    ! Character: ^
    PROC char_caret(\num nScaleParam)
        VAR robtarget pTarget;
        VAR num nScale:=1;
        pTarget:=refTarget;
        IF Present(nScaleParam) THEN
            nScale:=nScaleParam;
        ENDIF
        pTarget.trans:=[8*nScale,34.0*nScale,0];
        MoveL pTarget,vSpeed,fine,tTool\WObj:=wWobj;
        Set do_pen;
        pTarget.trans:=[0*nScale,20.0*nScale,0];
        MoveL pTarget,vSpeed,fine,tTool\WObj:=wWobj;
        Reset do_pen;
        MoveL RelTool(pTarget,0,0,-2),vSpeed,z0,tTool\WObj:=wWobj;
        pTarget.trans:=[8*nScale,34.0*nScale,0];
        MoveL pTarget,vSpeed,fine,tTool\WObj:=wWobj;
        Set do_pen;
        pTarget.trans:=[16*nScale,20.0*nScale,0];
        MoveL pTarget,vSpeed,fine,tTool\WObj:=wWobj;
        Reset do_pen;
        MoveL RelTool(pTarget,0,0,-2),vSpeed,z0,tTool\WObj:=wWobj;
        wWobj.oframe.trans.x:=wWobj.oframe.trans.x+16*nScale;
    ENDPROC

    ! Character: &
    PROC char_ampersand(\num nScaleParam)
        VAR robtarget pTarget;
        VAR num nScale:=1;
        pTarget:=refTarget;
        IF Present(nScaleParam) THEN
            nScale:=nScaleParam;
        ENDIF
        pTarget.trans:=[23*nScale,23.0*nScale,0];
        MoveL pTarget,vSpeed,fine,tTool\WObj:=wWobj;
        Set do_pen;
        pTarget.trans:=[23*nScale,24.0*nScale,0];
        MoveL pTarget,vSpeed,z0,tTool\WObj:=wWobj;
        pTarget.trans:=[22*nScale,25.0*nScale,0];
        MoveL pTarget,vSpeed,z0,tTool\WObj:=wWobj;
        pTarget.trans:=[21*nScale,25.0*nScale,0];
        MoveL pTarget,vSpeed,z0,tTool\WObj:=wWobj;
        pTarget.trans:=[20*nScale,24.0*nScale,0];
        MoveL pTarget,vSpeed,z0,tTool\WObj:=wWobj;
        pTarget.trans:=[19*nScale,22.0*nScale,0];
        MoveL pTarget,vSpeed,z0,tTool\WObj:=wWobj;
        pTarget.trans:=[17*nScale,17.0*nScale,0];
        MoveL pTarget,vSpeed,z0,tTool\WObj:=wWobj;
        pTarget.trans:=[15*nScale,14.0*nScale,0];
        MoveL pTarget,vSpeed,z0,tTool\WObj:=wWobj;
        pTarget.trans:=[13*nScale,12.0*nScale,0];
        MoveL pTarget,vSpeed,z0,tTool\WObj:=wWobj;
        pTarget.trans:=[11*nScale,11.0*nScale,0];
        MoveL pTarget,vSpeed,z0,tTool\WObj:=wWobj;
        pTarget.trans:=[7*nScale,11.0*nScale,0];
        MoveL pTarget,vSpeed,z0,tTool\WObj:=wWobj;
        pTarget.trans:=[5*nScale,12.0*nScale,0];
        MoveL pTarget,vSpeed,z0,tTool\WObj:=wWobj;
        pTarget.trans:=[4*nScale,13.0*nScale,0];
        MoveL pTarget,vSpeed,z0,tTool\WObj:=wWobj;
        pTarget.trans:=[3*nScale,15.0*nScale,0];
        MoveL pTarget,vSpeed,z0,tTool\WObj:=wWobj;
        pTarget.trans:=[3*nScale,17.0*nScale,0];
        MoveL pTarget,vSpeed,z0,tTool\WObj:=wWobj;
        pTarget.trans:=[4*nScale,19.0*nScale,0];
        MoveL pTarget,vSpeed,z0,tTool\WObj:=wWobj;
        pTarget.trans:=[5*nScale,20.0*nScale,0];
        MoveL pTarget,vSpeed,z0,tTool\WObj:=wWobj;
        pTarget.trans:=[12*nScale,24.0*nScale,0];
        MoveL pTarget,vSpeed,z0,tTool\WObj:=wWobj;
        pTarget.trans:=[13*nScale,25.0*nScale,0];
        MoveL pTarget,vSpeed,z0,tTool\WObj:=wWobj;
        pTarget.trans:=[14*nScale,27.0*nScale,0];
        MoveL pTarget,vSpeed,z0,tTool\WObj:=wWobj;
        pTarget.trans:=[14*nScale,29.0*nScale,0];
        MoveL pTarget,vSpeed,z0,tTool\WObj:=wWobj;
        pTarget.trans:=[13*nScale,31.0*nScale,0];
        MoveL pTarget,vSpeed,z0,tTool\WObj:=wWobj;
        pTarget.trans:=[11*nScale,32.0*nScale,0];
        MoveL pTarget,vSpeed,z0,tTool\WObj:=wWobj;
        pTarget.trans:=[9*nScale,31.0*nScale,0];
        MoveL pTarget,vSpeed,z0,tTool\WObj:=wWobj;
        pTarget.trans:=[8*nScale,29.0*nScale,0];
        MoveL pTarget,vSpeed,z0,tTool\WObj:=wWobj;
        pTarget.trans:=[8*nScale,27.0*nScale,0];
        MoveL pTarget,vSpeed,z0,tTool\WObj:=wWobj;
        pTarget.trans:=[9*nScale,24.0*nScale,0];
        MoveL pTarget,vSpeed,z0,tTool\WObj:=wWobj;
        pTarget.trans:=[11*nScale,21.0*nScale,0];
        MoveL pTarget,vSpeed,z0,tTool\WObj:=wWobj;
        pTarget.trans:=[16*nScale,14.0*nScale,0];
        MoveL pTarget,vSpeed,z0,tTool\WObj:=wWobj;
        pTarget.trans:=[18*nScale,12.0*nScale,0];
        MoveL pTarget,vSpeed,z0,tTool\WObj:=wWobj;
        pTarget.trans:=[20*nScale,11.0*nScale,0];
        MoveL pTarget,vSpeed,z0,tTool\WObj:=wWobj;
        pTarget.trans:=[22*nScale,11.0*nScale,0];
        MoveL pTarget,vSpeed,z0,tTool\WObj:=wWobj;
        pTarget.trans:=[23*nScale,12.0*nScale,0];
        MoveL pTarget,vSpeed,z0,tTool\WObj:=wWobj;
        pTarget.trans:=[23*nScale,13.0*nScale,0];
        MoveL pTarget,vSpeed,fine,tTool\WObj:=wWobj;
        Reset do_pen;
        MoveL RelTool(pTarget,0,0,-2),vSpeed,z0,tTool\WObj:=wWobj;
        wWobj.oframe.trans.x:=wWobj.oframe.trans.x+26*nScale;
    ENDPROC

    ! Character: *
    PROC char_asterisk(\num nScaleParam)
        VAR robtarget pTarget;
        VAR num nScale:=1;
        pTarget:=refTarget;
        IF Present(nScaleParam) THEN
            nScale:=nScaleParam;
        ENDIF
        pTarget.trans:=[8*nScale,26.0*nScale,0];
        MoveL pTarget,vSpeed,fine,tTool\WObj:=wWobj;
        Set do_pen;
        pTarget.trans:=[8*nScale,14.0*nScale,0];
        MoveL pTarget,vSpeed,fine,tTool\WObj:=wWobj;
        Reset do_pen;
        MoveL RelTool(pTarget,0,0,-2),vSpeed,z0,tTool\WObj:=wWobj;
        pTarget.trans:=[3*nScale,23.0*nScale,0];
        MoveL pTarget,vSpeed,fine,tTool\WObj:=wWobj;
        Set do_pen;
        pTarget.trans:=[13*nScale,17.0*nScale,0];
        MoveL pTarget,vSpeed,fine,tTool\WObj:=wWobj;
        Reset do_pen;
        MoveL RelTool(pTarget,0,0,-2),vSpeed,z0,tTool\WObj:=wWobj;
        pTarget.trans:=[13*nScale,23.0*nScale,0];
        MoveL pTarget,vSpeed,fine,tTool\WObj:=wWobj;
        Set do_pen;
        pTarget.trans:=[3*nScale,17.0*nScale,0];
        MoveL pTarget,vSpeed,fine,tTool\WObj:=wWobj;
        Reset do_pen;
        MoveL RelTool(pTarget,0,0,-2),vSpeed,z0,tTool\WObj:=wWobj;
        wWobj.oframe.trans.x:=wWobj.oframe.trans.x+16*nScale;
    ENDPROC

    ! Character: (
    PROC char_leftparenthesis(\num nScaleParam)
        VAR robtarget pTarget;
        VAR num nScale:=1;
        pTarget:=refTarget;
        IF Present(nScaleParam) THEN
            nScale:=nScaleParam;
        ENDIF
        pTarget.trans:=[11*nScale,36.0*nScale,0];
        MoveL pTarget,vSpeed,fine,tTool\WObj:=wWobj;
        Set do_pen;
        pTarget.trans:=[9*nScale,34.0*nScale,0];
        MoveL pTarget,vSpeed,z0,tTool\WObj:=wWobj;
        pTarget.trans:=[7*nScale,31.0*nScale,0];
        MoveL pTarget,vSpeed,z0,tTool\WObj:=wWobj;
        pTarget.trans:=[5*nScale,27.0*nScale,0];
        MoveL pTarget,vSpeed,z0,tTool\WObj:=wWobj;
        pTarget.trans:=[4*nScale,22.0*nScale,0];
        MoveL pTarget,vSpeed,z0,tTool\WObj:=wWobj;
        pTarget.trans:=[4*nScale,18.0*nScale,0];
        MoveL pTarget,vSpeed,z0,tTool\WObj:=wWobj;
        pTarget.trans:=[5*nScale,13.0*nScale,0];
        MoveL pTarget,vSpeed,z0,tTool\WObj:=wWobj;
        pTarget.trans:=[7*nScale,9.0*nScale,0];
        MoveL pTarget,vSpeed,z0,tTool\WObj:=wWobj;
        pTarget.trans:=[9*nScale,6.0*nScale,0];
        MoveL pTarget,vSpeed,z0,tTool\WObj:=wWobj;
        pTarget.trans:=[11*nScale,4.0*nScale,0];
        MoveL pTarget,vSpeed,fine,tTool\WObj:=wWobj;
        Reset do_pen;
        MoveL RelTool(pTarget,0,0,-2),vSpeed,z0,tTool\WObj:=wWobj;
        wWobj.oframe.trans.x:=wWobj.oframe.trans.x+14*nScale;
    ENDPROC

    ! Character: )
    PROC char_rightparenthesis(\num nScaleParam)
        VAR robtarget pTarget;
        VAR num nScale:=1;
        pTarget:=refTarget;
        IF Present(nScaleParam) THEN
            nScale:=nScaleParam;
        ENDIF
        pTarget.trans:=[3*nScale,36.0*nScale,0];
        MoveL pTarget,vSpeed,fine,tTool\WObj:=wWobj;
        Set do_pen;
        pTarget.trans:=[5*nScale,34.0*nScale,0];
        MoveL pTarget,vSpeed,z0,tTool\WObj:=wWobj;
        pTarget.trans:=[7*nScale,31.0*nScale,0];
        MoveL pTarget,vSpeed,z0,tTool\WObj:=wWobj;
        pTarget.trans:=[9*nScale,27.0*nScale,0];
        MoveL pTarget,vSpeed,z0,tTool\WObj:=wWobj;
        pTarget.trans:=[10*nScale,22.0*nScale,0];
        MoveL pTarget,vSpeed,z0,tTool\WObj:=wWobj;
        pTarget.trans:=[10*nScale,18.0*nScale,0];
        MoveL pTarget,vSpeed,z0,tTool\WObj:=wWobj;
        pTarget.trans:=[9*nScale,13.0*nScale,0];
        MoveL pTarget,vSpeed,z0,tTool\WObj:=wWobj;
        pTarget.trans:=[7*nScale,9.0*nScale,0];
        MoveL pTarget,vSpeed,z0,tTool\WObj:=wWobj;
        pTarget.trans:=[5*nScale,6.0*nScale,0];
        MoveL pTarget,vSpeed,z0,tTool\WObj:=wWobj;
        pTarget.trans:=[3*nScale,4.0*nScale,0];
        MoveL pTarget,vSpeed,fine,tTool\WObj:=wWobj;
        Reset do_pen;
        MoveL RelTool(pTarget,0,0,-2),vSpeed,z0,tTool\WObj:=wWobj;
        wWobj.oframe.trans.x:=wWobj.oframe.trans.x+14*nScale;
    ENDPROC

    ! Character: +
    PROC char_plus(\num nScaleParam)
        VAR robtarget pTarget;
        VAR num nScale:=1;
        pTarget:=refTarget;
        IF Present(nScaleParam) THEN
            nScale:=nScaleParam;
        ENDIF
        pTarget.trans:=[13*nScale,29.0*nScale,0];
        MoveL pTarget,vSpeed,fine,tTool\WObj:=wWobj;
        Set do_pen;
        pTarget.trans:=[13*nScale,11.0*nScale,0];
        MoveL pTarget,vSpeed,fine,tTool\WObj:=wWobj;
        Reset do_pen;
        MoveL RelTool(pTarget,0,0,-2),vSpeed,z0,tTool\WObj:=wWobj;
        pTarget.trans:=[4*nScale,20.0*nScale,0];
        MoveL pTarget,vSpeed,fine,tTool\WObj:=wWobj;
        Set do_pen;
        pTarget.trans:=[22*nScale,20.0*nScale,0];
        MoveL pTarget,vSpeed,fine,tTool\WObj:=wWobj;
        Reset do_pen;
        MoveL RelTool(pTarget,0,0,-2),vSpeed,z0,tTool\WObj:=wWobj;
        wWobj.oframe.trans.x:=wWobj.oframe.trans.x+26*nScale;
    ENDPROC

    ! Character: =
    PROC char_equals(\num nScaleParam)
        VAR robtarget pTarget;
        VAR num nScale:=1;
        pTarget:=refTarget;
        IF Present(nScaleParam) THEN
            nScale:=nScaleParam;
        ENDIF
        pTarget.trans:=[4*nScale,23.0*nScale,0];
        MoveL pTarget,vSpeed,fine,tTool\WObj:=wWobj;
        Set do_pen;
        pTarget.trans:=[22*nScale,23.0*nScale,0];
        MoveL pTarget,vSpeed,fine,tTool\WObj:=wWobj;
        Reset do_pen;
        MoveL RelTool(pTarget,0,0,-2),vSpeed,z0,tTool\WObj:=wWobj;
        pTarget.trans:=[4*nScale,17.0*nScale,0];
        MoveL pTarget,vSpeed,fine,tTool\WObj:=wWobj;
        Set do_pen;
        pTarget.trans:=[22*nScale,17.0*nScale,0];
        MoveL pTarget,vSpeed,fine,tTool\WObj:=wWobj;
        Reset do_pen;
        MoveL RelTool(pTarget,0,0,-2),vSpeed,z0,tTool\WObj:=wWobj;
        wWobj.oframe.trans.x:=wWobj.oframe.trans.x+26*nScale;
    ENDPROC

    ! Character: [
    PROC char_leftbracket(\num nScaleParam)
        VAR robtarget pTarget;
        VAR num nScale:=1;
        pTarget:=refTarget;
        IF Present(nScaleParam) THEN
            nScale:=nScaleParam;
        ENDIF
        pTarget.trans:=[4*nScale,36.0*nScale,0];
        MoveL pTarget,vSpeed,fine,tTool\WObj:=wWobj;
        Set do_pen;
        pTarget.trans:=[4*nScale,4.0*nScale,0];
        MoveL pTarget,vSpeed,fine,tTool\WObj:=wWobj;
        Reset do_pen;
        MoveL RelTool(pTarget,0,0,-2),vSpeed,z0,tTool\WObj:=wWobj;
        pTarget.trans:=[5*nScale,36.0*nScale,0];
        MoveL pTarget,vSpeed,fine,tTool\WObj:=wWobj;
        Set do_pen;
        pTarget.trans:=[5*nScale,4.0*nScale,0];
        MoveL pTarget,vSpeed,fine,tTool\WObj:=wWobj;
        Reset do_pen;
        MoveL RelTool(pTarget,0,0,-2),vSpeed,z0,tTool\WObj:=wWobj;
        pTarget.trans:=[4*nScale,36.0*nScale,0];
        MoveL pTarget,vSpeed,fine,tTool\WObj:=wWobj;
        Set do_pen;
        pTarget.trans:=[11*nScale,36.0*nScale,0];
        MoveL pTarget,vSpeed,fine,tTool\WObj:=wWobj;
        Reset do_pen;
        MoveL RelTool(pTarget,0,0,-2),vSpeed,z0,tTool\WObj:=wWobj;
        pTarget.trans:=[4*nScale,4.0*nScale,0];
        MoveL pTarget,vSpeed,fine,tTool\WObj:=wWobj;
        Set do_pen;
        pTarget.trans:=[11*nScale,4.0*nScale,0];
        MoveL pTarget,vSpeed,fine,tTool\WObj:=wWobj;
        Reset do_pen;
        MoveL RelTool(pTarget,0,0,-2),vSpeed,z0,tTool\WObj:=wWobj;
        wWobj.oframe.trans.x:=wWobj.oframe.trans.x+14*nScale;
    ENDPROC

    ! Character: ]
    PROC char_rightbracket(\num nScaleParam)
        VAR robtarget pTarget;
        VAR num nScale:=1;
        pTarget:=refTarget;
        IF Present(nScaleParam) THEN
            nScale:=nScaleParam;
        ENDIF
        pTarget.trans:=[9*nScale,36.0*nScale,0];
        MoveL pTarget,vSpeed,fine,tTool\WObj:=wWobj;
        Set do_pen;
        pTarget.trans:=[9*nScale,4.0*nScale,0];
        MoveL pTarget,vSpeed,fine,tTool\WObj:=wWobj;
        Reset do_pen;
        MoveL RelTool(pTarget,0,0,-2),vSpeed,z0,tTool\WObj:=wWobj;
        pTarget.trans:=[10*nScale,36.0*nScale,0];
        MoveL pTarget,vSpeed,fine,tTool\WObj:=wWobj;
        Set do_pen;
        pTarget.trans:=[10*nScale,4.0*nScale,0];
        MoveL pTarget,vSpeed,fine,tTool\WObj:=wWobj;
        Reset do_pen;
        MoveL RelTool(pTarget,0,0,-2),vSpeed,z0,tTool\WObj:=wWobj;
        pTarget.trans:=[3*nScale,36.0*nScale,0];
        MoveL pTarget,vSpeed,fine,tTool\WObj:=wWobj;
        Set do_pen;
        pTarget.trans:=[10*nScale,36.0*nScale,0];
        MoveL pTarget,vSpeed,fine,tTool\WObj:=wWobj;
        Reset do_pen;
        MoveL RelTool(pTarget,0,0,-2),vSpeed,z0,tTool\WObj:=wWobj;
        pTarget.trans:=[3*nScale,4.0*nScale,0];
        MoveL pTarget,vSpeed,fine,tTool\WObj:=wWobj;
        Set do_pen;
        pTarget.trans:=[10*nScale,4.0*nScale,0];
        MoveL pTarget,vSpeed,fine,tTool\WObj:=wWobj;
        Reset do_pen;
        MoveL RelTool(pTarget,0,0,-2),vSpeed,z0,tTool\WObj:=wWobj;
        wWobj.oframe.trans.x:=wWobj.oframe.trans.x+14*nScale;
    ENDPROC

    ! Character: {
    PROC char_leftbrace(\num nScaleParam)
        VAR robtarget pTarget;
        VAR num nScale:=1;
        pTarget:=refTarget;
        IF Present(nScaleParam) THEN
            nScale:=nScaleParam;
        ENDIF
        pTarget.trans:=[9*nScale,36.0*nScale,0];
        MoveL pTarget,vSpeed,fine,tTool\WObj:=wWobj;
        Set do_pen;
        pTarget.trans:=[7*nScale,35.0*nScale,0];
        MoveL pTarget,vSpeed,z0,tTool\WObj:=wWobj;
        pTarget.trans:=[6*nScale,34.0*nScale,0];
        MoveL pTarget,vSpeed,z0,tTool\WObj:=wWobj;
        pTarget.trans:=[5*nScale,32.0*nScale,0];
        MoveL pTarget,vSpeed,z0,tTool\WObj:=wWobj;
        pTarget.trans:=[5*nScale,30.0*nScale,0];
        MoveL pTarget,vSpeed,z0,tTool\WObj:=wWobj;
        pTarget.trans:=[6*nScale,28.0*nScale,0];
        MoveL pTarget,vSpeed,z0,tTool\WObj:=wWobj;
        pTarget.trans:=[7*nScale,27.0*nScale,0];
        MoveL pTarget,vSpeed,z0,tTool\WObj:=wWobj;
        pTarget.trans:=[8*nScale,25.0*nScale,0];
        MoveL pTarget,vSpeed,z0,tTool\WObj:=wWobj;
        pTarget.trans:=[8*nScale,23.0*nScale,0];
        MoveL pTarget,vSpeed,z0,tTool\WObj:=wWobj;
        pTarget.trans:=[6*nScale,21.0*nScale,0];
        MoveL pTarget,vSpeed,fine,tTool\WObj:=wWobj;
        Reset do_pen;
        MoveL RelTool(pTarget,0,0,-2),vSpeed,z0,tTool\WObj:=wWobj;
        pTarget.trans:=[7*nScale,35.0*nScale,0];
        MoveL pTarget,vSpeed,fine,tTool\WObj:=wWobj;
        Set do_pen;
        pTarget.trans:=[6*nScale,33.0*nScale,0];
        MoveL pTarget,vSpeed,z0,tTool\WObj:=wWobj;
        pTarget.trans:=[6*nScale,31.0*nScale,0];
        MoveL pTarget,vSpeed,z0,tTool\WObj:=wWobj;
        pTarget.trans:=[7*nScale,29.0*nScale,0];
        MoveL pTarget,vSpeed,z0,tTool\WObj:=wWobj;
        pTarget.trans:=[8*nScale,28.0*nScale,0];
        MoveL pTarget,vSpeed,z0,tTool\WObj:=wWobj;
        pTarget.trans:=[9*nScale,26.0*nScale,0];
        MoveL pTarget,vSpeed,z0,tTool\WObj:=wWobj;
        pTarget.trans:=[9*nScale,24.0*nScale,0];
        MoveL pTarget,vSpeed,z0,tTool\WObj:=wWobj;
        pTarget.trans:=[8*nScale,22.0*nScale,0];
        MoveL pTarget,vSpeed,z0,tTool\WObj:=wWobj;
        pTarget.trans:=[4*nScale,20.0*nScale,0];
        MoveL pTarget,vSpeed,z0,tTool\WObj:=wWobj;
        pTarget.trans:=[8*nScale,18.0*nScale,0];
        MoveL pTarget,vSpeed,z0,tTool\WObj:=wWobj;
        pTarget.trans:=[9*nScale,16.0*nScale,0];
        MoveL pTarget,vSpeed,z0,tTool\WObj:=wWobj;
        pTarget.trans:=[9*nScale,14.0*nScale,0];
        MoveL pTarget,vSpeed,z0,tTool\WObj:=wWobj;
        pTarget.trans:=[8*nScale,12.0*nScale,0];
        MoveL pTarget,vSpeed,z0,tTool\WObj:=wWobj;
        pTarget.trans:=[7*nScale,11.0*nScale,0];
        MoveL pTarget,vSpeed,z0,tTool\WObj:=wWobj;
        pTarget.trans:=[6*nScale,9.0*nScale,0];
        MoveL pTarget,vSpeed,z0,tTool\WObj:=wWobj;
        pTarget.trans:=[6*nScale,7.0*nScale,0];
        MoveL pTarget,vSpeed,z0,tTool\WObj:=wWobj;
        pTarget.trans:=[7*nScale,5.0*nScale,0];
        MoveL pTarget,vSpeed,fine,tTool\WObj:=wWobj;
        Reset do_pen;
        MoveL RelTool(pTarget,0,0,-2),vSpeed,z0,tTool\WObj:=wWobj;
        pTarget.trans:=[6*nScale,19.0*nScale,0];
        MoveL pTarget,vSpeed,fine,tTool\WObj:=wWobj;
        Set do_pen;
        pTarget.trans:=[8*nScale,17.0*nScale,0];
        MoveL pTarget,vSpeed,z0,tTool\WObj:=wWobj;
        pTarget.trans:=[8*nScale,15.0*nScale,0];
        MoveL pTarget,vSpeed,z0,tTool\WObj:=wWobj;
        pTarget.trans:=[7*nScale,13.0*nScale,0];
        MoveL pTarget,vSpeed,z0,tTool\WObj:=wWobj;
        pTarget.trans:=[6*nScale,12.0*nScale,0];
        MoveL pTarget,vSpeed,z0,tTool\WObj:=wWobj;
        pTarget.trans:=[5*nScale,10.0*nScale,0];
        MoveL pTarget,vSpeed,z0,tTool\WObj:=wWobj;
        pTarget.trans:=[5*nScale,8.0*nScale,0];
        MoveL pTarget,vSpeed,z0,tTool\WObj:=wWobj;
        pTarget.trans:=[6*nScale,6.0*nScale,0];
        MoveL pTarget,vSpeed,z0,tTool\WObj:=wWobj;
        pTarget.trans:=[7*nScale,5.0*nScale,0];
        MoveL pTarget,vSpeed,z0,tTool\WObj:=wWobj;
        pTarget.trans:=[9*nScale,4.0*nScale,0];
        MoveL pTarget,vSpeed,fine,tTool\WObj:=wWobj;
        Reset do_pen;
        MoveL RelTool(pTarget,0,0,-2),vSpeed,z0,tTool\WObj:=wWobj;
        wWobj.oframe.trans.x:=wWobj.oframe.trans.x+14*nScale;
    ENDPROC

    ! Character: }
    PROC char_rightbrace(\num nScaleParam)
        VAR robtarget pTarget;
        VAR num nScale:=1;
        pTarget:=refTarget;
        IF Present(nScaleParam) THEN
            nScale:=nScaleParam;
        ENDIF
        pTarget.trans:=[5*nScale,36.0*nScale,0];
        MoveL pTarget,vSpeed,fine,tTool\WObj:=wWobj;
        Set do_pen;
        pTarget.trans:=[7*nScale,35.0*nScale,0];
        MoveL pTarget,vSpeed,z0,tTool\WObj:=wWobj;
        pTarget.trans:=[8*nScale,34.0*nScale,0];
        MoveL pTarget,vSpeed,z0,tTool\WObj:=wWobj;
        pTarget.trans:=[9*nScale,32.0*nScale,0];
        MoveL pTarget,vSpeed,z0,tTool\WObj:=wWobj;
        pTarget.trans:=[9*nScale,30.0*nScale,0];
        MoveL pTarget,vSpeed,z0,tTool\WObj:=wWobj;
        pTarget.trans:=[8*nScale,28.0*nScale,0];
        MoveL pTarget,vSpeed,z0,tTool\WObj:=wWobj;
        pTarget.trans:=[7*nScale,27.0*nScale,0];
        MoveL pTarget,vSpeed,z0,tTool\WObj:=wWobj;
        pTarget.trans:=[6*nScale,25.0*nScale,0];
        MoveL pTarget,vSpeed,z0,tTool\WObj:=wWobj;
        pTarget.trans:=[6*nScale,23.0*nScale,0];
        MoveL pTarget,vSpeed,z0,tTool\WObj:=wWobj;
        pTarget.trans:=[8*nScale,21.0*nScale,0];
        MoveL pTarget,vSpeed,fine,tTool\WObj:=wWobj;
        Reset do_pen;
        MoveL RelTool(pTarget,0,0,-2),vSpeed,z0,tTool\WObj:=wWobj;
        pTarget.trans:=[7*nScale,35.0*nScale,0];
        MoveL pTarget,vSpeed,fine,tTool\WObj:=wWobj;
        Set do_pen;
        pTarget.trans:=[8*nScale,33.0*nScale,0];
        MoveL pTarget,vSpeed,z0,tTool\WObj:=wWobj;
        pTarget.trans:=[8*nScale,31.0*nScale,0];
        MoveL pTarget,vSpeed,z0,tTool\WObj:=wWobj;
        pTarget.trans:=[7*nScale,29.0*nScale,0];
        MoveL pTarget,vSpeed,z0,tTool\WObj:=wWobj;
        pTarget.trans:=[6*nScale,28.0*nScale,0];
        MoveL pTarget,vSpeed,z0,tTool\WObj:=wWobj;
        pTarget.trans:=[5*nScale,26.0*nScale,0];
        MoveL pTarget,vSpeed,z0,tTool\WObj:=wWobj;
        pTarget.trans:=[5*nScale,24.0*nScale,0];
        MoveL pTarget,vSpeed,z0,tTool\WObj:=wWobj;
        pTarget.trans:=[6*nScale,22.0*nScale,0];
        MoveL pTarget,vSpeed,z0,tTool\WObj:=wWobj;
        pTarget.trans:=[10*nScale,20.0*nScale,0];
        MoveL pTarget,vSpeed,z0,tTool\WObj:=wWobj;
        pTarget.trans:=[6*nScale,18.0*nScale,0];
        MoveL pTarget,vSpeed,z0,tTool\WObj:=wWobj;
        pTarget.trans:=[5*nScale,16.0*nScale,0];
        MoveL pTarget,vSpeed,z0,tTool\WObj:=wWobj;
        pTarget.trans:=[5*nScale,14.0*nScale,0];
        MoveL pTarget,vSpeed,z0,tTool\WObj:=wWobj;
        pTarget.trans:=[6*nScale,12.0*nScale,0];
        MoveL pTarget,vSpeed,z0,tTool\WObj:=wWobj;
        pTarget.trans:=[7*nScale,11.0*nScale,0];
        MoveL pTarget,vSpeed,z0,tTool\WObj:=wWobj;
        pTarget.trans:=[8*nScale,9.0*nScale,0];
        MoveL pTarget,vSpeed,z0,tTool\WObj:=wWobj;
        pTarget.trans:=[8*nScale,7.0*nScale,0];
        MoveL pTarget,vSpeed,z0,tTool\WObj:=wWobj;
        pTarget.trans:=[7*nScale,5.0*nScale,0];
        MoveL pTarget,vSpeed,fine,tTool\WObj:=wWobj;
        Reset do_pen;
        MoveL RelTool(pTarget,0,0,-2),vSpeed,z0,tTool\WObj:=wWobj;
        pTarget.trans:=[8*nScale,19.0*nScale,0];
        MoveL pTarget,vSpeed,fine,tTool\WObj:=wWobj;
        Set do_pen;
        pTarget.trans:=[6*nScale,17.0*nScale,0];
        MoveL pTarget,vSpeed,z0,tTool\WObj:=wWobj;
        pTarget.trans:=[6*nScale,15.0*nScale,0];
        MoveL pTarget,vSpeed,z0,tTool\WObj:=wWobj;
        pTarget.trans:=[7*nScale,13.0*nScale,0];
        MoveL pTarget,vSpeed,z0,tTool\WObj:=wWobj;
        pTarget.trans:=[8*nScale,12.0*nScale,0];
        MoveL pTarget,vSpeed,z0,tTool\WObj:=wWobj;
        pTarget.trans:=[9*nScale,10.0*nScale,0];
        MoveL pTarget,vSpeed,z0,tTool\WObj:=wWobj;
        pTarget.trans:=[9*nScale,8.0*nScale,0];
        MoveL pTarget,vSpeed,z0,tTool\WObj:=wWobj;
        pTarget.trans:=[8*nScale,6.0*nScale,0];
        MoveL pTarget,vSpeed,z0,tTool\WObj:=wWobj;
        pTarget.trans:=[7*nScale,5.0*nScale,0];
        MoveL pTarget,vSpeed,z0,tTool\WObj:=wWobj;
        pTarget.trans:=[5*nScale,4.0*nScale,0];
        MoveL pTarget,vSpeed,fine,tTool\WObj:=wWobj;
        Reset do_pen;
        MoveL RelTool(pTarget,0,0,-2),vSpeed,z0,tTool\WObj:=wWobj;
        wWobj.oframe.trans.x:=wWobj.oframe.trans.x+14*nScale;
    ENDPROC

    ! Character: |
    PROC char_pipe(\num nScaleParam)
        VAR robtarget pTarget;
        VAR num nScale:=1;
        pTarget:=refTarget;
        IF Present(nScaleParam) THEN
            nScale:=nScaleParam;
        ENDIF
        pTarget.trans:=[4*nScale,36.0*nScale,0];
        MoveL pTarget,vSpeed,fine,tTool\WObj:=wWobj;
        Set do_pen;
        pTarget.trans:=[4*nScale,4.0*nScale,0];
        MoveL pTarget,vSpeed,fine,tTool\WObj:=wWobj;
        Reset do_pen;
        MoveL RelTool(pTarget,0,0,-2),vSpeed,z0,tTool\WObj:=wWobj;
        wWobj.oframe.trans.x:=wWobj.oframe.trans.x+8*nScale;
    ENDPROC

    ! Character: <
    PROC char_lessthan(\num nScaleParam)
        VAR robtarget pTarget;
        VAR num nScale:=1;
        pTarget:=refTarget;
        IF Present(nScaleParam) THEN
            nScale:=nScaleParam;
        ENDIF
        pTarget.trans:=[20*nScale,29.0*nScale,0];
        MoveL pTarget,vSpeed,fine,tTool\WObj:=wWobj;
        Set do_pen;
        pTarget.trans:=[4*nScale,20.0*nScale,0];
        MoveL pTarget,vSpeed,z0,tTool\WObj:=wWobj;
        pTarget.trans:=[20*nScale,11.0*nScale,0];
        MoveL pTarget,vSpeed,fine,tTool\WObj:=wWobj;
        Reset do_pen;
        MoveL RelTool(pTarget,0,0,-2),vSpeed,z0,tTool\WObj:=wWobj;
        wWobj.oframe.trans.x:=wWobj.oframe.trans.x+24*nScale;
    ENDPROC

    ! Character: >
    PROC char_greaterthan(\num nScaleParam)
        VAR robtarget pTarget;
        VAR num nScale:=1;
        pTarget:=refTarget;
        IF Present(nScaleParam) THEN
            nScale:=nScaleParam;
        ENDIF
        pTarget.trans:=[4*nScale,29.0*nScale,0];
        MoveL pTarget,vSpeed,fine,tTool\WObj:=wWobj;
        Set do_pen;
        pTarget.trans:=[20*nScale,20.0*nScale,0];
        MoveL pTarget,vSpeed,z0,tTool\WObj:=wWobj;
        pTarget.trans:=[4*nScale,11.0*nScale,0];
        MoveL pTarget,vSpeed,fine,tTool\WObj:=wWobj;
        Reset do_pen;
        MoveL RelTool(pTarget,0,0,-2),vSpeed,z0,tTool\WObj:=wWobj;
        wWobj.oframe.trans.x:=wWobj.oframe.trans.x+24*nScale;
    ENDPROC

    ! Character: ?
    PROC char_question(\num nScaleParam)
        VAR robtarget pTarget;
        VAR num nScale:=1;
        pTarget:=refTarget;
        IF Present(nScaleParam) THEN
            nScale:=nScaleParam;
        ENDIF
        pTarget.trans:=[3*nScale,27.0*nScale,0];
        MoveL pTarget,vSpeed,fine,tTool\WObj:=wWobj;
        Set do_pen;
        pTarget.trans:=[3*nScale,28.0*nScale,0];
        MoveL pTarget,vSpeed,z0,tTool\WObj:=wWobj;
        pTarget.trans:=[4*nScale,30.0*nScale,0];
        MoveL pTarget,vSpeed,z0,tTool\WObj:=wWobj;
        pTarget.trans:=[5*nScale,31.0*nScale,0];
        MoveL pTarget,vSpeed,z0,tTool\WObj:=wWobj;
        pTarget.trans:=[7*nScale,32.0*nScale,0];
        MoveL pTarget,vSpeed,z0,tTool\WObj:=wWobj;
        pTarget.trans:=[11*nScale,32.0*nScale,0];
        MoveL pTarget,vSpeed,z0,tTool\WObj:=wWobj;
        pTarget.trans:=[13*nScale,31.0*nScale,0];
        MoveL pTarget,vSpeed,z0,tTool\WObj:=wWobj;
        pTarget.trans:=[14*nScale,30.0*nScale,0];
        MoveL pTarget,vSpeed,z0,tTool\WObj:=wWobj;
        pTarget.trans:=[15*nScale,28.0*nScale,0];
        MoveL pTarget,vSpeed,z0,tTool\WObj:=wWobj;
        pTarget.trans:=[15*nScale,26.0*nScale,0];
        MoveL pTarget,vSpeed,z0,tTool\WObj:=wWobj;
        pTarget.trans:=[14*nScale,24.0*nScale,0];
        MoveL pTarget,vSpeed,z0,tTool\WObj:=wWobj;
        pTarget.trans:=[13*nScale,23.0*nScale,0];
        MoveL pTarget,vSpeed,z0,tTool\WObj:=wWobj;
        pTarget.trans:=[9*nScale,21.0*nScale,0];
        MoveL pTarget,vSpeed,z0,tTool\WObj:=wWobj;
        pTarget.trans:=[9*nScale,18.0*nScale,0];
        MoveL pTarget,vSpeed,fine,tTool\WObj:=wWobj;
        Reset do_pen;
        MoveL RelTool(pTarget,0,0,-2),vSpeed,z0,tTool\WObj:=wWobj;
        pTarget.trans:=[9*nScale,13.0*nScale,0];
        MoveL pTarget,vSpeed,fine,tTool\WObj:=wWobj;
        Set do_pen;
        pTarget.trans:=[8*nScale,12.0*nScale,0];
        MoveL pTarget,vSpeed,z0,tTool\WObj:=wWobj;
        pTarget.trans:=[9*nScale,11.0*nScale,0];
        MoveL pTarget,vSpeed,z0,tTool\WObj:=wWobj;
        pTarget.trans:=[10*nScale,12.0*nScale,0];
        MoveL pTarget,vSpeed,z0,tTool\WObj:=wWobj;
        pTarget.trans:=[9*nScale,13.0*nScale,0];
        MoveL pTarget,vSpeed,fine,tTool\WObj:=wWobj;
        Reset do_pen;
        MoveL RelTool(pTarget,0,0,-2),vSpeed,z0,tTool\WObj:=wWobj;
        wWobj.oframe.trans.x:=wWobj.oframe.trans.x+18*nScale;
    ENDPROC

    ! Character: _
    PROC char_underscore(\num nScaleParam)
        VAR robtarget pTarget;
        VAR num nScale:=1;
        pTarget:=refTarget;
        IF Present(nScaleParam) THEN
            nScale:=nScaleParam;
        ENDIF
        pTarget.trans:=[0*nScale,4.0*nScale,0];
        MoveL pTarget,vSpeed,fine,tTool\WObj:=wWobj;
        Set do_pen;
        pTarget.trans:=[20*nScale,4.0*nScale,0];
        MoveL pTarget,vSpeed,fine,tTool\WObj:=wWobj;
        Reset do_pen;
        MoveL RelTool(pTarget,0,0,-2),vSpeed,z0,tTool\WObj:=wWobj;
        wWobj.oframe.trans.x:=wWobj.oframe.trans.x+20*nScale;
    ENDPROC

    ! Character: -
    PROC char_minus(\num nScaleParam)
        VAR robtarget pTarget;
        VAR num nScale:=1;
        pTarget:=refTarget;
        IF Present(nScaleParam) THEN
            nScale:=nScaleParam;
        ENDIF
        pTarget.trans:=[4*nScale,20.0*nScale,0];
        MoveL pTarget,vSpeed,fine,tTool\WObj:=wWobj;
        Set do_pen;
        pTarget.trans:=[22*nScale,20.0*nScale,0];
        MoveL pTarget,vSpeed,fine,tTool\WObj:=wWobj;
        Reset do_pen;
        MoveL RelTool(pTarget,0,0,-2),vSpeed,z0,tTool\WObj:=wWobj;
        wWobj.oframe.trans.x:=wWobj.oframe.trans.x+26*nScale;
    ENDPROC

    ! Character: ~
    PROC char_tilde(\num nScaleParam)
        VAR robtarget pTarget;
        VAR num nScale:=1;
        pTarget:=refTarget;
        IF Present(nScaleParam) THEN
            nScale:=nScaleParam;
        ENDIF
        pTarget.trans:=[3*nScale,17.0*nScale,0];
        MoveL pTarget,vSpeed,fine,tTool\WObj:=wWobj;
        Set do_pen;
        pTarget.trans:=[3*nScale,19.0*nScale,0];
        MoveL pTarget,vSpeed,z0,tTool\WObj:=wWobj;
        pTarget.trans:=[4*nScale,22.0*nScale,0];
        MoveL pTarget,vSpeed,z0,tTool\WObj:=wWobj;
        pTarget.trans:=[6*nScale,23.0*nScale,0];
        MoveL pTarget,vSpeed,z0,tTool\WObj:=wWobj;
        pTarget.trans:=[8*nScale,23.0*nScale,0];
        MoveL pTarget,vSpeed,z0,tTool\WObj:=wWobj;
        pTarget.trans:=[10*nScale,22.0*nScale,0];
        MoveL pTarget,vSpeed,z0,tTool\WObj:=wWobj;
        pTarget.trans:=[14*nScale,19.0*nScale,0];
        MoveL pTarget,vSpeed,z0,tTool\WObj:=wWobj;
        pTarget.trans:=[16*nScale,18.0*nScale,0];
        MoveL pTarget,vSpeed,z0,tTool\WObj:=wWobj;
        pTarget.trans:=[18*nScale,18.0*nScale,0];
        MoveL pTarget,vSpeed,z0,tTool\WObj:=wWobj;
        pTarget.trans:=[20*nScale,19.0*nScale,0];
        MoveL pTarget,vSpeed,z0,tTool\WObj:=wWobj;
        pTarget.trans:=[21*nScale,21.0*nScale,0];
        MoveL pTarget,vSpeed,fine,tTool\WObj:=wWobj;
        Reset do_pen;
        MoveL RelTool(pTarget,0,0,-2),vSpeed,z0,tTool\WObj:=wWobj;
        pTarget.trans:=[3*nScale,19.0*nScale,0];
        MoveL pTarget,vSpeed,fine,tTool\WObj:=wWobj;
        Set do_pen;
        pTarget.trans:=[4*nScale,21.0*nScale,0];
        MoveL pTarget,vSpeed,z0,tTool\WObj:=wWobj;
        pTarget.trans:=[6*nScale,22.0*nScale,0];
        MoveL pTarget,vSpeed,z0,tTool\WObj:=wWobj;
        pTarget.trans:=[8*nScale,22.0*nScale,0];
        MoveL pTarget,vSpeed,z0,tTool\WObj:=wWobj;
        pTarget.trans:=[10*nScale,21.0*nScale,0];
        MoveL pTarget,vSpeed,z0,tTool\WObj:=wWobj;
        pTarget.trans:=[14*nScale,18.0*nScale,0];
        MoveL pTarget,vSpeed,z0,tTool\WObj:=wWobj;
        pTarget.trans:=[16*nScale,17.0*nScale,0];
        MoveL pTarget,vSpeed,z0,tTool\WObj:=wWobj;
        pTarget.trans:=[18*nScale,17.0*nScale,0];
        MoveL pTarget,vSpeed,z0,tTool\WObj:=wWobj;
        pTarget.trans:=[20*nScale,18.0*nScale,0];
        MoveL pTarget,vSpeed,z0,tTool\WObj:=wWobj;
        pTarget.trans:=[21*nScale,21.0*nScale,0];
        MoveL pTarget,vSpeed,z0,tTool\WObj:=wWobj;
        pTarget.trans:=[21*nScale,23.0*nScale,0];
        MoveL pTarget,vSpeed,fine,tTool\WObj:=wWobj;
        Reset do_pen;
        MoveL RelTool(pTarget,0,0,-2),vSpeed,z0,tTool\WObj:=wWobj;
        wWobj.oframe.trans.x:=wWobj.oframe.trans.x+24*nScale;
    ENDPROC

    ! Character: .
    PROC char_period(\num nScaleParam)
        VAR robtarget pTarget;
        VAR num nScale:=1;
        pTarget:=refTarget;
        IF Present(nScaleParam) THEN
            nScale:=nScaleParam;
        ENDIF
        pTarget.trans:=[4*nScale,16.0*nScale,0];
        MoveL pTarget,vSpeed,fine,tTool\WObj:=wWobj;
        Set do_pen;
        pTarget.trans:=[3*nScale,15.0*nScale,0];
        MoveL pTarget,vSpeed,z0,tTool\WObj:=wWobj;
        pTarget.trans:=[4*nScale,14.0*nScale,0];
        MoveL pTarget,vSpeed,z0,tTool\WObj:=wWobj;
        pTarget.trans:=[5*nScale,15.0*nScale,0];
        MoveL pTarget,vSpeed,z0,tTool\WObj:=wWobj;
        pTarget.trans:=[4*nScale,16.0*nScale,0];
        MoveL pTarget,vSpeed,fine,tTool\WObj:=wWobj;
        Reset do_pen;
        MoveL RelTool(pTarget,0,0,-2),vSpeed,z0,tTool\WObj:=wWobj;
        wWobj.oframe.trans.x:=wWobj.oframe.trans.x+8*nScale;
    ENDPROC

    ! Character: ,
    PROC char_comma(\num nScaleParam)
        VAR robtarget pTarget;
        VAR num nScale:=1;
        pTarget:=refTarget;
        IF Present(nScaleParam) THEN
            nScale:=nScaleParam;
        ENDIF
        pTarget.trans:=[5*nScale,15.0*nScale,0];
        MoveL pTarget,vSpeed,fine,tTool\WObj:=wWobj;
        Set do_pen;
        pTarget.trans:=[4*nScale,14.0*nScale,0];
        MoveL pTarget,vSpeed,z0,tTool\WObj:=wWobj;
        pTarget.trans:=[3*nScale,15.0*nScale,0];
        MoveL pTarget,vSpeed,z0,tTool\WObj:=wWobj;
        pTarget.trans:=[4*nScale,16.0*nScale,0];
        MoveL pTarget,vSpeed,z0,tTool\WObj:=wWobj;
        pTarget.trans:=[5*nScale,15.0*nScale,0];
        MoveL pTarget,vSpeed,z0,tTool\WObj:=wWobj;
        pTarget.trans:=[5*nScale,13.0*nScale,0];
        MoveL pTarget,vSpeed,z0,tTool\WObj:=wWobj;
        pTarget.trans:=[3*nScale,11.0*nScale,0];
        MoveL pTarget,vSpeed,fine,tTool\WObj:=wWobj;
        Reset do_pen;
        MoveL RelTool(pTarget,0,0,-2),vSpeed,z0,tTool\WObj:=wWobj;
        wWobj.oframe.trans.x:=wWobj.oframe.trans.x+8*nScale;
    ENDPROC

    ! Character: ;
    PROC char_semicolon(\num nScaleParam)
        VAR robtarget pTarget;
        VAR num nScale:=1;
        pTarget:=refTarget;
        IF Present(nScaleParam) THEN
            nScale:=nScaleParam;
        ENDIF
        pTarget.trans:=[4*nScale,23.0*nScale,0];
        MoveL pTarget,vSpeed,fine,tTool\WObj:=wWobj;
        Set do_pen;
        pTarget.trans:=[3*nScale,22.0*nScale,0];
        MoveL pTarget,vSpeed,z0,tTool\WObj:=wWobj;
        pTarget.trans:=[4*nScale,21.0*nScale,0];
        MoveL pTarget,vSpeed,z0,tTool\WObj:=wWobj;
        pTarget.trans:=[5*nScale,22.0*nScale,0];
        MoveL pTarget,vSpeed,z0,tTool\WObj:=wWobj;
        pTarget.trans:=[4*nScale,23.0*nScale,0];
        MoveL pTarget,vSpeed,fine,tTool\WObj:=wWobj;
        Reset do_pen;
        MoveL RelTool(pTarget,0,0,-2),vSpeed,z0,tTool\WObj:=wWobj;
        pTarget.trans:=[5*nScale,15.0*nScale,0];
        MoveL pTarget,vSpeed,fine,tTool\WObj:=wWobj;
        Set do_pen;
        pTarget.trans:=[4*nScale,14.0*nScale,0];
        MoveL pTarget,vSpeed,z0,tTool\WObj:=wWobj;
        pTarget.trans:=[3*nScale,15.0*nScale,0];
        MoveL pTarget,vSpeed,z0,tTool\WObj:=wWobj;
        pTarget.trans:=[4*nScale,16.0*nScale,0];
        MoveL pTarget,vSpeed,z0,tTool\WObj:=wWobj;
        pTarget.trans:=[5*nScale,15.0*nScale,0];
        MoveL pTarget,vSpeed,z0,tTool\WObj:=wWobj;
        pTarget.trans:=[5*nScale,13.0*nScale,0];
        MoveL pTarget,vSpeed,z0,tTool\WObj:=wWobj;
        pTarget.trans:=[3*nScale,11.0*nScale,0];
        MoveL pTarget,vSpeed,fine,tTool\WObj:=wWobj;
        Reset do_pen;
        MoveL RelTool(pTarget,0,0,-2),vSpeed,z0,tTool\WObj:=wWobj;
        wWobj.oframe.trans.x:=wWobj.oframe.trans.x+8*nScale;
    ENDPROC

    ! Character: :
    PROC char_colon(\num nScaleParam)
        VAR robtarget pTarget;
        VAR num nScale:=1;
        pTarget:=refTarget;
        IF Present(nScaleParam) THEN
            nScale:=nScaleParam;
        ENDIF
        pTarget.trans:=[4*nScale,23.0*nScale,0];
        MoveL pTarget,vSpeed,fine,tTool\WObj:=wWobj;
        Set do_pen;
        pTarget.trans:=[3*nScale,22.0*nScale,0];
        MoveL pTarget,vSpeed,z0,tTool\WObj:=wWobj;
        pTarget.trans:=[4*nScale,21.0*nScale,0];
        MoveL pTarget,vSpeed,z0,tTool\WObj:=wWobj;
        pTarget.trans:=[5*nScale,22.0*nScale,0];
        MoveL pTarget,vSpeed,z0,tTool\WObj:=wWobj;
        pTarget.trans:=[4*nScale,23.0*nScale,0];
        MoveL pTarget,vSpeed,fine,tTool\WObj:=wWobj;
        Reset do_pen;
        MoveL RelTool(pTarget,0,0,-2),vSpeed,z0,tTool\WObj:=wWobj;
        pTarget.trans:=[4*nScale,16.0*nScale,0];
        MoveL pTarget,vSpeed,fine,tTool\WObj:=wWobj;
        Set do_pen;
        pTarget.trans:=[3*nScale,15.0*nScale,0];
        MoveL pTarget,vSpeed,z0,tTool\WObj:=wWobj;
        pTarget.trans:=[4*nScale,14.0*nScale,0];
        MoveL pTarget,vSpeed,z0,tTool\WObj:=wWobj;
        pTarget.trans:=[5*nScale,15.0*nScale,0];
        MoveL pTarget,vSpeed,z0,tTool\WObj:=wWobj;
        pTarget.trans:=[4*nScale,16.0*nScale,0];
        MoveL pTarget,vSpeed,fine,tTool\WObj:=wWobj;
        Reset do_pen;
        MoveL RelTool(pTarget,0,0,-2),vSpeed,z0,tTool\WObj:=wWobj;
        wWobj.oframe.trans.x:=wWobj.oframe.trans.x+8*nScale;
    ENDPROC
ENDMODULE

--- Controller Data/IRB1200_5_90/RAPID/TASK1/PROGMOD/Module1.modx ---
MODULE Module1
    PERS tooldata tTool:=[TRUE,[[110,0,140],[0.707106781,0,0.707106781,0]],[1,[10.7435139,0,140],[1,0,0,0],0,0,0]];
    PERS wobjdata wWobj:=[FALSE,TRUE,"",[[526.92,-115.652,257.517],[0.695575,0.127182,0.127182,0.695575]],[[769,100,1],[1,0,0,0]]];
    VAR speeddata vSpeed:=[300,3000,100,3000];
    PERS tooldata Pen_TCP:=[TRUE,[[110,0,140],[0.707106781,0,0.707106781,0]],[1,[10.7435139,0,140],[1,0,0,0],0,0,0]];
    CONST robtarget refTarget:=[[-61.41097207,14.187566617,-0.240748359],[0.098541688,-0.538960856,-0.836538911,-0.00365808],[-1,-1,0,1],[9E+09,9E+09,9E+09,9E+09,9E+09,9E+09]];

    PROC main()
        VAR robtarget pNow;
        reset do_pen;
        wWobj.oframe.trans.z:=1;
        wWobj.oframe.trans.y:=150;
        wWobj.oframe.trans.x:=wobj0.oframe.trans.x+20;
        WriteCursive "the quick brown fox jumps over the lazy dog"\nScaleParam:=0.5;
        reset do_pen;
        wWobj.oframe.trans.z:=1;
        wWobj.oframe.trans.y:=100;
        wWobj.oframe.trans.x:=wobj0.oframe.trans.x+20;
        WriteCursive "THE QUICK BROWN FOX JUMPS OVER THE LAZY DOG";
        pNow:=CRobT();
        MoveL RelTool(pNow,0,0,-40),vmax,fine,tTool\wobj:=wWobj;
    ENDPROC

    PROC writeCursive(string sText,\num nScaleParam)
        VAR num i;
        VAR string sChar;
        VAR num nScale:=1;
        IF Present(nScaleParam) THEN
            nScale:=nScaleParam;
        ENDIF
        FOR i FROM 1 TO StrLen(sText) DO
            sChar:=StrPart(sText,i,1);
            TEST sChar
            CASE "a":
                char_a\nScaleParam:=nScale;
            CASE "b":
                char_b\nScaleParam:=nScale;
            CASE "c":
                char_c\nScaleParam:=nScale;
            CASE "d":
                char_d\nScaleParam:=nScale;
            CASE "e":
                char_e\nScaleParam:=nScale;
            CASE "f":
                char_f\nScaleParam:=nScale;
            CASE "g":
                char_g\nScaleParam:=nScale;
            CASE "h":
                char_h\nScaleParam:=nScale;
            CASE "i":
                char_i\nScaleParam:=nScale;
            CASE "j":
                char_j\nScaleParam:=nScale;
            CASE "k":
                char_k\nScaleParam:=nScale;
            CASE "l":
                char_l\nScaleParam:=nScale;
            CASE "m":
                char_m\nScaleParam:=nScale;
            CASE "n":
                char_n\nScaleParam:=nScale;
            CASE "o":
                char_o\nScaleParam:=nScale;
            CASE "p":
                char_p\nScaleParam:=nScale;
            CASE "q":
                char_q\nScaleParam:=nScale;
            CASE "r":
                char_r\nScaleParam:=nScale;
            CASE "s":
                char_s\nScaleParam:=nScale;
            CASE "t":
                char_t\nScaleParam:=nScale;
            CASE "u":
                char_u\nScaleParam:=nScale;
            CASE "v":
                char_v\nScaleParam:=nScale;
            CASE "w":
                char_w\nScaleParam:=nScale;
            CASE "x":
                char_x\nScaleParam:=nScale;
            CASE "y":
                char_y\nScaleParam:=nScale;
            CASE "z":
                char_z\nScaleParam:=nScale;
            CASE "A":
                char_upperA\nScaleParam:=nScale;
            CASE "B":
                char_upperB\nScaleParam:=nScale;
            CASE "C":
                char_upperC\nScaleParam:=nScale;
            CASE "D":
                char_upperD\nScaleParam:=nScale;
            CASE "E":
                char_upperE\nScaleParam:=nScale;
            CASE "F":
                char_upperF\nScaleParam:=nScale;
            CASE "G":
                char_upperG\nScaleParam:=nScale;
            CASE "H":
                char_upperH\nScaleParam:=nScale;
            CASE "I":
                char_upperI\nScaleParam:=nScale;
            CASE "J":
                char_upperJ\nScaleParam:=nScale;
            CASE "K":
                char_upperK\nScaleParam:=nScale;
            CASE "L":
                char_upperL\nScaleParam:=nScale;
            CASE "M":
                char_upperM\nScaleParam:=nScale;
            CASE "N":
                char_upperN\nScaleParam:=nScale;
            CASE "O":
                char_upperO\nScaleParam:=nScale;
            CASE "P":
                char_upperP\nScaleParam:=nScale;
            CASE "Q":
                char_upperQ\nScaleParam:=nScale;
            CASE "R":
                char_upperR\nScaleParam:=nScale;
            CASE "S":
                char_upperS\nScaleParam:=nScale;
            CASE "T":
                char_upperT\nScaleParam:=nScale;
            CASE "U":
                char_upperU\nScaleParam:=nScale;
            CASE "V":
                char_upperV\nScaleParam:=nScale;
            CASE "W":
                char_upperW\nScaleParam:=nScale;
            CASE "X":
                char_upperX\nScaleParam:=nScale;
            CASE "Y":
                char_upperY\nScaleParam:=nScale;
            CASE "Z":
                char_upperZ\nScaleParam:=nScale;
            CASE "0":
                char_0\nScaleParam:=nScale;
            CASE "1":
                char_1\nScaleParam:=nScale;
            CASE "2":
                char_2\nScaleParam:=nScale;
            CASE "3":
                char_3\nScaleParam:=nScale;
            CASE "4":
                char_4\nScaleParam:=nScale;
            CASE "5":
                char_5\nScaleParam:=nScale;
            CASE "6":
                char_6\nScaleParam:=nScale;
            CASE "7":
                char_7\nScaleParam:=nScale;
            CASE "8":
                char_8\nScaleParam:=nScale;
            CASE "9":
                char_9\nScaleParam:=nScale;
            CASE "!":
                char_exclamation\nScaleParam:=nScale;
            CASE "@":
                char_at\nScaleParam:=nScale;
            CASE "#":
                char_hash\nScaleParam:=nScale;
            CASE "$":
                char_dollar\nScaleParam:=nScale;
            CASE "%":
                char_percent\nScaleParam:=nScale;
            CASE "^":
                char_caret\nScaleParam:=nScale;
            CASE "&":
                char_ampersand\nScaleParam:=nScale;
            CASE "*":
                char_asterisk\nScaleParam:=nScale;
            CASE "(":
                char_leftparenthesis\nScaleParam:=nScale;
            CASE ")":
                char_rightparenthesis\nScaleParam:=nScale;
            CASE "+":
                char_plus\nScaleParam:=nScale;
            CASE "=":
                char_equals\nScaleParam:=nScale;
            CASE "[":
                char_leftbracket\nScaleParam:=nScale;
            CASE "]":
                char_rightbracket\nScaleParam:=nScale;
            CASE "{":
                char_leftbrace\nScaleParam:=nScale;
            CASE "}":
                char_rightbrace\nScaleParam:=nScale;
            CASE "|":
                char_pipe\nScaleParam:=nScale;
            CASE "<":
                char_lessthan\nScaleParam:=nScale;
            CASE ">":
                char_greaterthan\nScaleParam:=nScale;
            CASE "?":
                char_question\nScaleParam:=nScale;
            CASE "_":
                char_underscore\nScaleParam:=nScale;
            CASE "-":
                char_minus\nScaleParam:=nScale;
            CASE "~":
                char_tilde\nScaleParam:=nScale;
            CASE ".":
                char_period\nScaleParam:=nScale;
            CASE ",":
                char_comma\nScaleParam:=nScale;
            CASE ";":
                char_semicolon\nScaleParam:=nScale;
            CASE ":":
                char_colon\nScaleParam:=nScale;
            CASE " ":
                ! Space - move right without drawing wWobj.oframe.trans.x:=wWobj.oframe.trans.x+15*nScale;
            DEFAULT:
                TPWrite "Character not supported: "+sChar;
            ENDTEST
        ENDFOR
    ENDPROC
ENDMODULE

--- Controller Data/IRB1200_5_90/SYSPAR/EIO.cfg ---
EIO:CFG_1.0:7:0::
#
VIRTUAL_NETWORK:

      -Name "Virtual" -Label "Virtual Device Network"
#
EIO_SIGNAL:

      -Name "IIO_di1" -SignalType "DI" -Device "IntegratedIOInternalDevice"\
      -DeviceMap "0"

      -Name "IIO_di2" -SignalType "DI" -Device "IntegratedIOInternalDevice"\
      -DeviceMap "1"

      -Name "IIO_di3" -SignalType "DI" -Device "IntegratedIOInternalDevice"\
      -DeviceMap "2"

      -Name "IIO_di4" -SignalType "DI" -Device "IntegratedIOInternalDevice"\
      -DeviceMap "3"

      -Name "IIO_di5" -SignalType "DI" -Device "IntegratedIOInternalDevice"\
      -DeviceMap "4"

      -Name "IIO_di6" -SignalType "DI" -Device "IntegratedIOInternalDevice"\
      -DeviceMap "5"

      -Name "IIO_di7" -SignalType "DI" -Device "IntegratedIOInternalDevice"\
      -DeviceMap "6"

      -Name "IIO_di8" -SignalType "DI" -Device "IntegratedIOInternalDevice"\
      -DeviceMap "7"

      -Name "IIO_di9" -SignalType "DI" -Device "IntegratedIOInternalDevice"\
      -DeviceMap "8"

      -Name "IIO_di10" -SignalType "DI" -Device "IntegratedIOInternalDevice"\
      -DeviceMap "9"

      -Name "IIO_di11" -SignalType "DI" -Device "IntegratedIOInternalDevice"\
      -DeviceMap "10"

      -Name "IIO_di12" -SignalType "DI" -Device "IntegratedIOInternalDevice"\
      -DeviceMap "11"

      -Name "IIO_di13" -SignalType "DI" -Device "IntegratedIOInternalDevice"\
      -DeviceMap "12"

      -Name "IIO_di14" -SignalType "DI" -Device "IntegratedIOInternalDevice"\
      -DeviceMap "13"

      -Name "IIO_di15" -SignalType "DI" -Device "IntegratedIOInternalDevice"\
      -DeviceMap "14"

      -Name "IIO_di16" -SignalType "DI" -Device "IntegratedIOInternalDevice"\
      -DeviceMap "15"

      -Name "IIO_do1" -SignalType "DO" -Device "IntegratedIOInternalDevice"\
      -DeviceMap "0"

      -Name "IIO_do2" -SignalType "DO" -Device "IntegratedIOInternalDevice"\
      -DeviceMap "1"

      -Name "IIO_do3" -SignalType "DO" -Device "IntegratedIOInternalDevice"\
      -DeviceMap "2"

      -Name "IIO_do4" -SignalType "DO" -Device "IntegratedIOInternalDevice"\
      -DeviceMap "3"

      -Name "IIO_do5" -SignalType "DO" -Device "IntegratedIOInternalDevice"\
      -DeviceMap "4"

      -Name "IIO_do6" -SignalType "DO" -Device "IntegratedIOInternalDevice"\
      -DeviceMap "5"

      -Name "IIO_do7" -SignalType "DO" -Device "IntegratedIOInternalDevice"\
      -DeviceMap "6"

      -Name "IIO_do8" -SignalType "DO" -Device "IntegratedIOInternalDevice"\
      -DeviceMap "7"

      -Name "IIO_gi" -SignalType "GI" -Device "integratedIOInternalDevice"\
      -DeviceMap "0-15"

      -Name "IIO_go" -SignalType "GO" -Device "integratedIOInternalDevice"\
      -DeviceMap "0-7"

      -Name "do_pen" -SignalType "DO" -Access "All"

#CTRL_SIGNATURE:UpI3rsGsdjPUEdBBGvNwuUTXFijTMgTtD42mLhnlGZgDW7Y00ZW5+aDJae9I93WBev467PSv26CaKbAkbr5rXw==

--- Controller Data/IRB1200_5_90/SYSPAR/PROC.cfg ---
PROC:CFG_1.0:7:0::

#CTRL_SIGNATURE:EanoTt332vqhZPmKvdzBrByTheeXv3GTX9o65SYsnrJ+DJbQQ2h+v49xbjzxd2tjmmEe4Rias40o22ORGzDJ/w==
